TYPE STRUCT_CM_Motor :
STRUCT
	CS	: CM_Motor_CS;
	HMI	: CM_Motor_HMI;
	STS	: CM_Motor_STS;
	ALM	: CM_Motor_ALM;
	WRN	: CM_Motor_WRN;
	PAR	: CM_Motor_PAR;
	SIM	: CM_Motor_SIM;
END_STRUCT
END_TYPE

(* stored: Version 1.1.0.1, ProductVersion 3.1.4024.12
   DUT STRUCT_CM_Motor: Id {da976e32-8b86-492c-9084-df13b160fb93} *)
